TYPE ST_Gear : //
STRUCT
	bEnable		                        :BOOL;	
	bGearOutMode                 :BOOL;
 
	bReady                            :BOOL;  
	bInGear		 	                   :BOOL;	
	bError				               :BOOL;			
END_STRUCT
END_TYPE

(* stored: Version 1.1.0.1, ProductVersion 3.1.4024.9
   DUT ST_Gear: Id {8a85ba3b-7aee-4f82-81c5-53787a6316f0} *)
